PROGRAM MAIN
VAR
END_VAR

PRG_DIAGNOSTIC();
PRG_SXR_VAC();

END_PROGRAM

(* stored: Version 1.1.0.1, ProductVersion 3.1.4022.16
   POU MAIN: Id {16be0fc6-ae40-4a05-90aa-9d2fd038dc01}, SpecialFunc None *)
